(* PLC project Generated.project, CODESYS CODESYS V3.5 SP19 Patch 1 *)
(* stored: creationDateTime 2026-09-15T02:12:09.700363, modificationDateTime 2026-09-15T02:12:09.700363 *)

(* ======================================================================= 🪜 ST_SpeedStepTable — Table des paliers de vitesse contacteurs ─────────────────────────────────────────────────────────────── 🎯 Rôle : Structure de configuration des contacteurs et seuils par palier 📄 Doc métier : DOC/AF/AF_Partie-10_Fonction_Winch_v2.1.md ======================================================================= *)
TYPE ST_SpeedStepTable : STRUCT
  P1R1 : BOOL;  (* === PALIER 1 (VITESSE MINIMALE) === Contacteur 1 pour Palier 1 *)
  P1R2 : BOOL;  (* Contacteur 2 pour Palier 1 *)
  P1R3 : BOOL;  (* Contacteur 3 pour Palier 1 *)
  P1R4 : BOOL;  (* Contacteur 4 pour Palier 1 *)
  P2R1 : BOOL;  (* === PALIER 2 === Contacteur 1 pour Palier 2 *)
  P2R2 : BOOL;  (* Contacteur 2 pour Palier 2 *)
  P2R3 : BOOL;  (* Contacteur 3 pour Palier 2 *)
  P2R4 : BOOL;  (* Contacteur 4 pour Palier 2 *)
  P3R1 : BOOL;  (* === PALIER 3 === Contacteur 1 pour Palier 3 *)
  P3R2 : BOOL;  (* Contacteur 2 pour Palier 3 *)
  P3R3 : BOOL;  (* Contacteur 3 pour Palier 3 *)
  P3R4 : BOOL;  (* Contacteur 4 pour Palier 3 *)
  P4R1 : BOOL;  (* === PALIER 4 === Contacteur 1 pour Palier 4 *)
  P4R2 : BOOL;  (* Contacteur 2 pour Palier 4 *)
  P4R3 : BOOL;  (* Contacteur 3 pour Palier 4 *)
  P4R4 : BOOL;  (* Contacteur 4 pour Palier 4 *)
  P5R1 : BOOL;  (* === PALIER 5 (VITESSE MAXIMALE) === Contacteur 1 pour Palier 5 *)
  P5R2 : BOOL;  (* Contacteur 2 pour Palier 5 *)
  P5R3 : BOOL;  (* Contacteur 3 pour Palier 5 *)
  P5R4 : BOOL;  (* Contacteur 4 pour Palier 5 *)
  StepThreshold_Pct : ARRAY[1..5] OF REAL;  (* === SEUILS DE TRANSITION (%) === Seuils de changement de palier (0..100%) *)
END_STRUCT;
END_TYPE

(* ======================================================================= 🔀 ST_SyncContactorDiag — Diagnostic discordance contacteurs M1/M2 ─────────────────────────────────────────────────────────────── 🎯 Rôle : dire EN CLAIR quel contacteur diverge entre M1 et M2 et à quel niveau on est (aucun / mismatch confirmé / escalade). Consommé par le bandeau IHM et le troubleshooting pour répondre « pourquoi ça bloque ». 🔒 Bits nommés (pas de masque hexa, AF03 §4). Plusieurs bits peuvent être TRUE simultanément (toutes les divergences détectées). 📄 Doc : DOC/AF/AF_Partie-10_Fonction_Winch_v2.1.md ======================================================================= *)
TYPE ST_SyncContactorDiag : STRUCT
  RelayFwdMismatch : BOOL;  (* TRUE = relais montée M1 <> M2 *)
  RelayRevMismatch : BOOL;  (* TRUE = relais descente M1 <> M2 *)
  Step1Mismatch : BOOL;  (* TRUE = contacteur palier 1 M1 <> M2 *)
  Step2Mismatch : BOOL;  (* TRUE = contacteur palier 2 M1 <> M2 *)
  Step3Mismatch : BOOL;  (* TRUE = contacteur palier 3 M1 <> M2 *)
  Step4Mismatch : BOOL;  (* TRUE = contacteur palier 4 M1 <> M2 *)
  MismatchLevel : INT;  (* 0 = aucun · 1 = discordance confirmée (SafeStop) · 2 = escalade (PowerCutOff) *)
END_STRUCT;
END_TYPE

(* ======================================================================= 🔀 FB_SyncContactor — Coherence commandes/contacteurs M1/M2 ─────────────────────────────────────────────────────────────── 🎯 Rôle : Detecter une discordance entre les commandes/contacteurs des 2 treuils (sens + paliers). Independante des codeurs — surveillable meme si les codeurs sont bypasses. 🔌 Interface : Bloc de surveillance transverse (1..N instances : requetes amont dans FB_WinchSync, sorties physiques finales dans PRG_06). 🔒 Polarite : ContactorMismatch = TRUE si discordance confirmee (debounce). Reponse GRADUEE : ContactorMismatch (niveau 1, filtre MismatchDebounce) -> SafeStop ; ContactorMismatchEscalated (niveau 2, si la discordance tient CST_SyncEscalationTime) -> escalade PowerCutOff. ⚖️ Concordance ACTIVE des que les 2 treuils sont commandes (relais ou contacteur) OU en mode synchronisme (SyncEnable). Seul BypassGlobal neutralise. 📄 Doc : DOC/AF/AF_Partie-10_Fonction_Winch_v2.1.md ======================================================================= *)
FUNCTION_BLOCK FB_SyncContactor
  VAR_INPUT
    Enable : BOOL;  (* === COMMANDES ET CONSIGNES === --> [CMD] Validation surveillance globale *)
    Reset : BOOL;  (* --> [CMD] Acquittement defaut sur front *)
    SyncEnable : BOOL;  (* --> [CMD] Autorisation utilisateur synchro *)
    RelayFwdM1 : BOOL;  (* === COMMANDES ET FEEDBACKS ACTIONS === --> [HW] Feedback/Ordre montee M1 *)
    RelayFwdM2 : BOOL;  (* --> [HW] Feedback/Ordre montee M2 *)
    RelayRevM1 : BOOL;  (* --> [HW] Feedback/Ordre descente M1 *)
    RelayRevM2 : BOOL;  (* --> [HW] Feedback/Ordre descente M2 *)
    Contactor1_M1 : BOOL;  (* --> [HW] Contacteur palier 1 M1 *)
    Contactor1_M2 : BOOL;  (* --> [HW] Contacteur palier 1 M2 *)
    Contactor2_M1 : BOOL;  (* --> [HW] Contacteur palier 2 M1 *)
    Contactor2_M2 : BOOL;  (* --> [HW] Contacteur palier 2 M2 *)
    Contactor3_M1 : BOOL;  (* --> [HW] Contacteur palier 3 M1 *)
    Contactor3_M2 : BOOL;  (* --> [HW] Contacteur palier 3 M2 *)
    Contactor4_M1 : BOOL;  (* --> [HW] Contacteur palier 4 M1 *)
    Contactor4_M2 : BOOL;  (* --> [HW] Contacteur palier 4 M2 *)
    BypassGlobal : BOOL := FALSE;  (* === BYPASSES ET SIMULATION === --> [TST] Neutralise la surveillance contacteurs *)
    DescentStep45Permit : BOOL := FALSE;  (* --> [CMD] Autorise uniquement le profil descente M1=P4 / M2=P5 *)
    SpeedStepTable : ST_SpeedStepTable;  (* --> [CFG] Table officielle paliers -> contacteurs *)
  END_VAR
  VAR_OUTPUT
    ContactorMismatch : BOOL;  (* === RESULTAT (reponse graduee) === <-- [SAFE] Niveau 1 : discordance commande/contacteurs confirmee (debounce) -> SafeStop *)
    ContactorMismatchEscalated : BOOL;  (* <-- [SAFE] Niveau 2 : discordance persistante -> escalade PowerCutOff *)
    CommandsCoherent : BOOL;  (* <-- [STAT] TRUE si le vecteur instantane est coherent ou derogation T291-A exacte *)
    DescentStep45Matched : BOOL;  (* <-- [STAT] TRUE si le profil M1=P4 / M2=P5 est exactement reconnu *)
    Diag : ST_SyncContactorDiag;  (* <-- [DIAG] Detail : quel contacteur diverge + niveau atteint *)
  END_VAR
  VAR
    MismatchDebounce : TIME := TIME#500ms;  (* Filtre transitoires/rampes avant de confirmer la discordance (niveau 1) *)
    CST_SyncEscalationTime : TIME := TIME#3s0ms;  (* Discordance confirmee tenue au-dela de ce delai -> escalade (niveau 2) *)
    MismatchTimer : TON;  (* === DETECTEURS ET TIMERS INTERNES === . [LOC] Tempo filtrage incoherence (niveau 1) *)
    EscalationTimer : TON;  (* . [LOC] Tempo escalade (niveau 2) *)
    MismatchActive : BOOL;  (* === VARIABLES LOCALES INTERNES === . [LOC] Discordance instantanee (avant debounce) *)
    BothCommanded : BOOL;  (* . [LOC] Les 2 treuils sont commandes (relais ou contacteur) *)
    DescentStep4M1 : BOOL;  (* . [LOC] M1 en descente avec vecteur table P4 exact *)
    DescentStep5M2 : BOOL;  (* . [LOC] M2 en descente avec vecteur table P5 exact *)
  END_VAR

            

{region "§1 Gate neutralisation"}
// 🛑 1. GATE
IF NOT Enable OR BypassGlobal THEN
    ContactorMismatch := FALSE;
    ContactorMismatchEscalated := FALSE;
    CommandsCoherent := FALSE;
    DescentStep45Matched := FALSE;
    MismatchActive := FALSE;
    BothCommanded := FALSE;
    DescentStep4M1 := FALSE;
    DescentStep5M2 := FALSE;
    MismatchTimer(IN := FALSE);
    EscalationTimer(IN := FALSE);
    Diag.RelayFwdMismatch := FALSE;
    Diag.RelayRevMismatch := FALSE;
    Diag.Step1Mismatch := FALSE;
    Diag.Step2Mismatch := FALSE;
    Diag.Step3Mismatch := FALSE;
    Diag.Step4Mismatch := FALSE;
    Diag.MismatchLevel := 0;
    RETURN;
END_IF;
{endregion}

{region "§2 Detection discordance + diagnostic decode"}
// 🔍 2. COHÉRENCE DES COMMANDES SÉCURITÉ — verifie que les commandes envoyees
// aux deux treuils sont identiques (sens et contacteurs).
// Concordance ACTIVE des que les 2 treuils sont commandes (relais ou contacteur)
// OU en mode synchronisme (SyncEnable).
BothCommanded := (RelayFwdM1 OR RelayRevM1 OR Contactor1_M1 OR Contactor2_M1
                  OR Contactor3_M1 OR Contactor4_M1)
             AND (RelayFwdM2 OR RelayRevM2 OR Contactor1_M2 OR Contactor2_M2
                  OR Contactor3_M2 OR Contactor4_M2);

// Diagnostic decode : quel(s) contacteur(s) diverge(nt) (bits nommes, plusieurs possibles).
Diag.RelayFwdMismatch := (BothCommanded OR SyncEnable) AND (RelayFwdM1 <> RelayFwdM2);
Diag.RelayRevMismatch := (BothCommanded OR SyncEnable) AND (RelayRevM1 <> RelayRevM2);
Diag.Step1Mismatch    := (BothCommanded OR SyncEnable) AND (Contactor1_M1 <> Contactor1_M2);
Diag.Step2Mismatch    := (BothCommanded OR SyncEnable) AND (Contactor2_M1 <> Contactor2_M2);
Diag.Step3Mismatch    := (BothCommanded OR SyncEnable) AND (Contactor3_M1 <> Contactor3_M2);
Diag.Step4Mismatch    := (BothCommanded OR SyncEnable) AND (Contactor4_M1 <> Contactor4_M2);

DescentStep4M1 := RelayRevM1 AND NOT RelayFwdM1
                  AND (Contactor1_M1 = SpeedStepTable.P4R1)
                  AND (Contactor2_M1 = SpeedStepTable.P4R2)
                  AND (Contactor3_M1 = SpeedStepTable.P4R3)
                  AND (Contactor4_M1 = SpeedStepTable.P4R4);
DescentStep5M2 := RelayRevM2 AND NOT RelayFwdM2
                  AND (Contactor1_M2 = SpeedStepTable.P5R1)
                  AND (Contactor2_M2 = SpeedStepTable.P5R2)
                  AND (Contactor3_M2 = SpeedStepTable.P5R3)
                  AND (Contactor4_M2 = SpeedStepTable.P5R4);
DescentStep45Matched := DescentStep45Permit
                        AND NOT RelayFwdM2
                        AND NOT RelayFwdM1
                        AND DescentStep4M1
                        AND DescentStep5M2;

IF DescentStep45Matched THEN
    Diag.Step1Mismatch := FALSE;
    Diag.Step2Mismatch := FALSE;
    Diag.Step3Mismatch := FALSE;
    Diag.Step4Mismatch := FALSE;
END_IF;

MismatchActive := Diag.RelayFwdMismatch OR Diag.RelayRevMismatch
    OR Diag.Step1Mismatch OR Diag.Step2Mismatch
    OR Diag.Step3Mismatch OR Diag.Step4Mismatch;
CommandsCoherent := NOT MismatchActive;

// Niveau 1 : discordance confirmee apres MismatchDebounce.
MismatchTimer(IN := MismatchActive, PT := MismatchDebounce);
ContactorMismatch := MismatchTimer.Q;

// Niveau 2 : la discordance confirmee tient au-dela de CST_SyncEscalationTime.
EscalationTimer(IN := ContactorMismatch, PT := CST_SyncEscalationTime);
ContactorMismatchEscalated := EscalationTimer.Q;

// Niveau publie.
IF ContactorMismatchEscalated THEN
    Diag.MismatchLevel := 2;
ELSIF ContactorMismatch THEN
    Diag.MismatchLevel := 1;
ELSE
    Diag.MismatchLevel := 0;
END_IF;
{endregion}

          
END_FUNCTION_BLOCK
